{attribute 'qualified_only'}
VAR_GLOBAL
	myVeryFirstDatamanGVL 	: TcoCognexVision.TcoDatamanIO_v_5_x_x;
END_VAR

(* stored: Version 1.1.0.1, ProductVersion 3.1.4024.11
   GVL GVL: Id {da8cc0c7-7535-0851-1cda-a5d24616e132} *)
